(* CODESYS project 1003_xlh_stamp_button_switch_led_joystick_remote.project
   Description: Receives some incoming messages and echoes them with CAN-ID +1
   Company: 3S - Smart Software Solutions GmbH
   Version: 1.0.0.0
   Title: CAN Bus API Example
   Author: 3S - Smart Software Solutions GmbH

Project tree, tasks and I/O mapping:
  xLH_base : CODESYS Control for Raspberry Pi 64 SL, CODESYS, order no. 2302000009, version 4.18.0.0
    application app
      libraries: Standard, 3.5.18.0 (System); Util, 3.5.21.0 (System); VisuDialogs, * (System); Memory, * (3S - Smart Software Solutions GmbH); CmpBitmapPool, * (System); CAN API, 1.0.0.4 (CODESYS); MemoryUtils, * (3S - Smart Software Solutions GmbH)
      task MAIN_TASK (cyclic, interval 10 ms, priority 1) calls MAIN
      task ENIPScannerServiceTask (cyclic, interval t#20ms, priority 30) calls EtherNet_IP_Scanner.ServiceCycle
      task ENIPScannerIOTask (cyclic, interval t#10ms, priority 0) calls EtherNet_IP_Scanner.IOCycle
      program MAIN [ST]
      trace Trace_Switch_Joystick (task MAIN_TASK): MAIN.fX, MAIN.fY
    Ethernet : Ethernet, CODESYS, version 4.2.0.0
        settings: IPAddress = [192,168,1,251]; SubnetMask = [255,255,255,0]; GatewayAddress = [192,168,1,1]; MACAddress = [16#2C,16#CF,16#67,16#D7,16#DB,16#D5]; NetworkInterfaceName = 'wlan0'; NetworkInterfaceName = "wlan0"; SaveCommunicationSettings = FALSE; IPAddress = [192,168,0,2]; SubnetMask = [255,255,255,0]; GatewayAddress = [0,0,0,0]
      EtherNet_IP_Scanner : EtherNet/IP Scanner, CODESYS, order no. 1, version 4.8.0.0
        dummy_joystick : dummy_joystick, CODESYS, version Major Revision=16#1, Minor Revision = 16#1
            settings: INITIALIZED = TRUE; IP address of Target = [16#C0,16#A8,16#01,16#97]; Keying.Check Minor Revision = FALSE; RequiredConfigVersion = 50660864; Number of Connections = 1; Connection Settings.Requested packet intervall = 10000 µs; Connection Settings.Connection Application Type = 2; Connection Settings.OT Connection Parameters = 18434; Connection Settings.TO Connection Parameters = 18450; Connection Settings.Connection Flags = 1062; Connection Settings.Connection Path Size = 6; Connection Settings.Large OT Connection Parameters = 1207959554; Connection Settings.Large TO Connection Parameters = 1207959570; Heartbeat Multiplier = 1; Joystick_fX.ReadOnly = False; Joystick_fX.BitSize = 64; Joystick_fX.DataSize = 8; Joystick_fY.ReadOnly = False; Joystick_fY.BitSize = 64; Joystick_fY.DataSize = 8; Joystick_fX.Name = 'Joystick_fX'; Joystick_fX.HelpString = ''; Joystick_fX.ReadOnly = False; Joystick_fX.BitSize = 64; Joystick_fX.DataSize = 8; Joystick_fX.DataType = 'LREAL'; Joystick_fY.Name = 'Joystick_fY'; Joystick_fY.HelpString = ''; Joystick_fY.ReadOnly = False; Joystick_fY.BitSize = 64; Joystick_fY.DataSize = 8; Joystick_fY.DataType = 'LREAL'; ConfigVersion = 50660864
            input  app.MAIN.fX : LREAL  // Joystick_fX
            input  app.MAIN.fY : LREAL  // Joystick_fY
    SoftMotion General Axis Pool
      a_axis : SM_Drive_PosControl, CODESYS, order no. 1805, version 4.18.0.0
          settings: wDriveID = 4; dwRatioTechUnitsDenom = 101846; iRatioTechUnitsNum = -125; eRampType = 1; fSWMaxVelocity = 50; fSWMaxAcceleration = 100; fSWMaxDeceleration = 100; fSWMaxJerk = 1000; fSWLimitNegative = -1000.0; ScalingIncs = 814768; ScalingUnits = 1000; InvertDirection = TRUE; IsLinearMotor = TRUE; MaximumOutputVelocityInt = 40738; MinimumOutputVelocityInt = -40738; Kp = 0.05; MaxFollowingError = 5.0; EnableFollowingErrorCheck = TRUE; DeadTime = 3.0
      x_axis : SM_Drive_PosControl, CODESYS, order no. 1805, version 4.18.0.0
          settings: dwRatioTechUnitsDenom = 101846; iRatioTechUnitsNum = 125; eRampType = 1; fSWMaxVelocity = 50; fSWMaxAcceleration = 100; fSWMaxDeceleration = 100; fSWMaxJerk = 1000; fSWLimitNegative = -1000; ScalingIncs = 814768; ScalingUnits = 1000; IsLinearMotor = TRUE; MaximumOutputVelocityInt = 40738; MinimumOutputVelocityInt = -40738; Kp = 0.05; MaxFollowingError = 5.0; EnableFollowingErrorCheck = TRUE; DeadTime = 3.0
      y_axis : SM_Drive_PosControl, CODESYS, order no. 1805, version 4.18.0.0
          settings: wDriveID = 2; dwRatioTechUnitsDenom = 101846; iRatioTechUnitsNum = 125; eRampType = 1; fSWMaxVelocity = 50; fSWMaxAcceleration = 100; fSWMaxDeceleration = 100; fSWMaxJerk = 1000; fSWLimitNegative = -1000; ScalingIncs = 814768; ScalingUnits = 1000; IsLinearMotor = TRUE; MaximumOutputVelocityInt = 40738; MinimumOutputVelocityInt = -40738; Kp = 0.05; MaxFollowingError = 5.0; EnableFollowingErrorCheck = TRUE; DeadTime = 3.0
      z_axis : SM_Drive_PosControl, CODESYS, order no. 1805, version 4.18.0.0
          settings: wDriveID = 3; dwRatioTechUnitsDenom = 101846; iRatioTechUnitsNum = 125; eRampType = 1; fSWMaxVelocity = 50; fSWMaxAcceleration = 100; fSWMaxDeceleration = 100; fSWMaxJerk = 1000; fSWLimitNegative = -1000; ScalingIncs = 814768; ScalingUnits = 1000; IsLinearMotor = TRUE; MaximumOutputVelocityInt = 40738; MinimumOutputVelocityInt = -40738; Kp = 0.05; MaxFollowingError = 5.0; EnableFollowingErrorCheck = TRUE; DeadTime = 3.0
    GPIOs_A_B : GPIOs B+/Pi2, CODESYS, version 4.15.0.0
        unmapped channels: digital inputs (GPIO0..GPIO31), digital outputs (GPIO0..GPIO31)
    Onewire
    Camera device
      <Leer>
    SPI
    I²C
  libraries: VisuSymbols, 4.5.0.0 (System); DepictorBase, 1.2.0.0 (CODESYS)
  text list GlobalTextList
  5ce3da45-db07-42e7-a21c-a00fff4ed8f6|C:\Users\phe\Downloads\Musterloesung_FUP.PNG
*)

// xLH_base/app/MAIN
PROGRAM MAIN
VAR
fX: LREAL;
fY: LREAL;
fDummy: LREAL;
END_VAR

// OPCUA Server
// https://www.youtube.com/watch?v=8TFpZLJTCY4

// OPCUA Client with Data source Manager
// https://www.youtube.com/watch?v=VxUwXuBgfXM

fDummy := fX;
fDummy := fY;

END_PROGRAM
